// TIA Portal V17 export
// export: Created 2024-08-09T12:53:18.7303991Z, ExportSetting WithDefaults, DisplayName Totally Integrated Automation Portal, DisplayVersion V17 Update 7, DisplayName TIA Portal Openness, DisplayVersion V17 Update 7, DisplayName TIA Portal Version Control Interface, DisplayVersion V17, DisplayName STEP 7 Professional, DisplayVersion V17 Update 7, DisplayName STEP 7 Safety, DisplayVersion V17 Update 6, DisplayName WinCC Professional, DisplayVersion V17 Update 7
TYPE "S_DOSBENNE"
// stored: IsFailsafeCompliant false
   STRUCT
      Benne { S7_SetPoint := 'True'} : "S_Benne";
      Pt_Zs { S7_SetPoint := 'True'} : "S_Suivi_Dosage";
      Dos_Commun { S7_SetPoint := 'True'} : "S_Dosage_Commun";
      Dial_Def { S7_SetPoint := 'True'} : "S_DIALOG_DEF";
      Lst_Compo_Affich { S7_SetPoint := 'True'} : Array[0.."Nbr_Max_Compo"] of "Affich_Compo";
      Lst_Compos { S7_SetPoint := 'True'} : Array[0.."Nbr_Max_Compo"] of "S_Com_Fab";
      Lst_Taches_Att_Vidange { S7_SetPoint := 'True'} : Array[0.."T_MAX_AMONTAVAL"] of "S_TacheNiv";
      Etat_Vibreur : Int;
      Deb_Dos : Date_And_Time;
      Mem_Pesees : Real;
      Mob_Agit : USInt;
      Num_Benne : SInt;
      FgArretVidange : Bool;
      Fg_Compo_Trouv : Bool;
      Fg_Complement : Bool;
      Fg_Ctrl_Conf : Bool;
      Fg_Proc_Exec : Bool;
   END_STRUCT;
   // Benne.Benne_Sync[0..9] := -1;
END_TYPE
